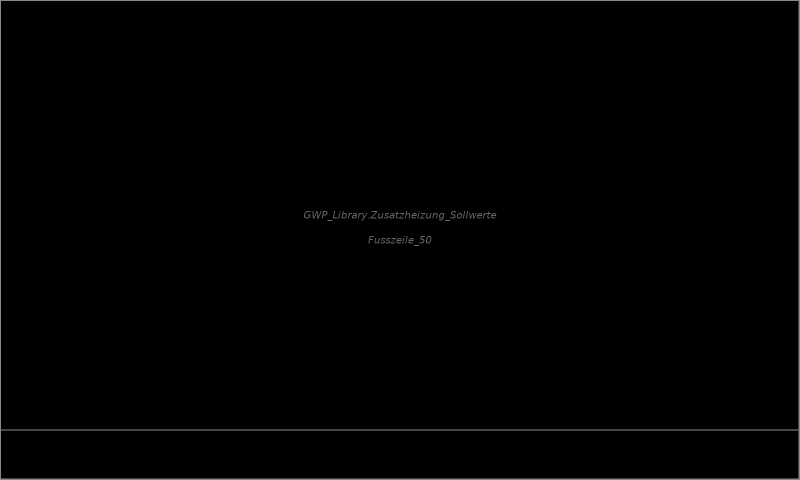
VISUALIZATION Zusatzheizung_Sollwerte  // 800x480
    Frame (0,0 800x430)
        shows GWP_Library.Zusatzheizung_Sollwerte(FB_Zusatzheizung := Main.Zusatzheizung_0)
    Frame (0,0 800x480)
        shows Fusszeile_50()
END_VISUALIZATION

(* stored: Version 1.1.0.1, ProductVersion 3.1.4022.6
   Visu Zusatzheizung_Sollwerte: Id {45e6dbc5-2d91-4c79-b3d7-a619cb7d3e91} *)
